# EPICS autosave request: iocBoot/obsolete/ioc13bmc_DAC_XPS/auto_settings.req
file "CARS_motor_settings.req",         P=$(P), M=m71
file "CARS_motor_settings.req",         P=$(P), M=m72
file "CARS_motor_settings.req",         P=$(P), M=m73
file "CARS_motor_settings.req",         P=$(P), M=m74
file "CARS_motor_settings.req",         P=$(P), M=m75
